FUNCTION_BLOCK FB_RRU7001
VAR_INPUT
END_VAR
VAR_OUTPUT
END_VAR
VAR
	fbNetwork       : FB_TcpClient; // Lắp động cơ mạng vào
    stTagData       : ST_RRU7001_Data; // Đem khuôn đúc ra hứng
    
    bInit           : BOOL := TRUE;
    bCardDetected   : BOOL;
END_VAR

// 1. CHẠY KHỞI TẠO 1 LẦN DUY NHẤT
IF bInit THEN
    fbNetwork.M_Connect(sIP_Address := '192.168.1.200', nPort := 20000); 
    bInit := FALSE;
END_IF

// 2. DUY TRÌ NHỊP ĐẬP CHO MẠNG TCP/IP (Gọi liên tục mỗi chu kỳ)
fbNetwork.M_Cyclic();

// 3. XỬ LÝ LOGIC QUÉT THẺ
IF fbNetwork.P_HasNewData THEN
    // Ép kiểu bằng MEMCPY
    fbNetwork.M_GetData(pDest := ADR(stTagData), nSize := SIZEOF(stTagData));
    
    bCardDetected := TRUE;
END_IF

END_FUNCTION_BLOCK

(* stored: Version 1.1.0.1, ProductVersion 3.1.4024.16
   POU FB_RRU7001: Id {76b6b341-bba7-4c91-a46d-1b0c622a711e}, SpecialFunc None *)
